// TIA Portal V20 export
DATA_BLOCK "LRemoteAccess_Data"   // DB275
TITLE = Data
AUTHOR : Siemens
// Storing data about mobile panel and UCP connection status
// stored: MemoryReserve 100
   VAR
      mobilePanel1 : "LRemoteAccess_typeMobilePanel";
      connectionBoxes : Array[1..2] of "LRemoteAccess_typeConnectionBox";
      ActivationMobileDP { S7_SetPoint := 'True'} : "LRemoteAccess_typeMobile_DeActivate";   // Activate Mobile Panel
      DeactivationMobileDP { S7_SetPoint := 'True'} : "LRemoteAccess_typeMobile_DeActivate";   // Deactivate Mobile Panel
      connectionTimeout { S7_SetPoint := 'True'} : Time := T#5s;   // Connection timeout. Keep greater than 3 sec. Default 5 sec.
   END_VAR
BEGIN
   connectionBoxes[1].ID := 20;
   connectionBoxes[2].ID := 21;
END_DATA_BLOCK
